// TIA Portal V17 export
// export: Created 2023-02-26T22:57:59.9998618Z, ExportSetting WithDefaults, DisplayName Totally Integrated Automation Portal, DisplayVersion V17, DisplayName TIA Portal Openness, DisplayVersion V17, DisplayName TIA Portal Version Control Interface, DisplayVersion V17, DisplayName TIA Portal Test Suite Advanced, DisplayVersion V17, DisplayName STEP 7 Professional, DisplayVersion V17, DisplayName SIMATIC Energy Suite, DisplayVersion V17, DisplayName STEP 7 Safety, DisplayVersion V17, DisplayName WinCC Professional, DisplayVersion V17
TYPE "stt_TimeWork"
// stored: IsFailsafeCompliant false
   STRUCT
      Seconds : USInt;
      Minute : USInt;
      Hours : USInt;
      Days : UDInt;
   END_STRUCT;
END_TYPE
